// TIA Portal project "Box Sorting" (V18)

(* hardware
DEVICE "S7-1200 station_1"  S7-1200 Station
   slot 0: "Rack_0"  S7-1200 Rack  Rack  V1.0
   slot 1: "PLC_1"  CPU 1212C AC/DC/Rly  6ES7 212-1BE40-0XB0  V4.6
*)

// ===== PLC "PLC_1"  CPU 1212C AC/DC/Rly =====

VAR_GLOBAL   // PLC tag table "Default tag table"
   "Start" AT %I0.0 : Bool;
   "Auto Mode" AT %M0.0 : Bool;
   "Stop" AT %I0.1 : Bool;
   "PE_Low" AT %I0.2 : Bool;
   "PE_High" AT %I0.3 : Bool;
   "#Large Box" AT %M0.1 : Bool;
   "Motor1" AT %Q0.0 : Bool;
   "Solenoid_valve" AT %Q0.1 : Bool;
   "Motor2" AT %Q0.2 : Bool;
   "num_L" AT %MW2 : Int;
   "num_S" AT %MW4 : Int;
   "total_box" AT %MW6 : Int;
   "num_L_real" AT %MD8 : Real;
   "num_S_real" AT %MD12 : Real;
   "total_box_real" AT %MD16 : Real;
   "percent_large" AT %MD20 : Real;
   "percent_small" AT %MD24 : Real;
   "Emergency Stop" AT %I0.4 : Bool;
END_VAR

// folder: System blocks/Program resources

DATA_BLOCK "timerA_DB"   // DB1
{ S7_Optimized_Access := 'TRUE' }
AUTHOR : Simatic
FAMILY : IEC
NAME : IEC_TMR
VERSION : 1.0
// stored: InstanceOfName IEC_TIMER
"IEC_TIMER"
BEGIN
END_DATA_BLOCK

DATA_BLOCK "timerB_DB"   // DB2
{ S7_Optimized_Access := 'TRUE' }
AUTHOR : Simatic
FAMILY : IEC
NAME : IEC_TMR
VERSION : 1.0
// stored: InstanceOfName IEC_TIMER
"IEC_TIMER"
BEGIN
END_DATA_BLOCK

DATA_BLOCK "timerC_DB"   // DB3
{ S7_Optimized_Access := 'TRUE' }
AUTHOR : Simatic
FAMILY : IEC
NAME : IEC_TMR
VERSION : 1.0
// stored: InstanceOfName IEC_TIMER
"IEC_TIMER"
BEGIN
END_DATA_BLOCK

DATA_BLOCK "timerD_DB"   // DB4
{ S7_Optimized_Access := 'TRUE' }
AUTHOR : Simatic
FAMILY : IEC
NAME : IEC_TMR
VERSION : 1.0
// stored: InstanceOfName IEC_TIMER
"IEC_TIMER"
BEGIN
END_DATA_BLOCK

DATA_BLOCK "CounterL_DB"   // DB5
{ S7_Optimized_Access := 'TRUE' }
AUTHOR : Simatic
FAMILY : IEC
NAME : CNTR
VERSION : 1.0
// stored: InstanceOfName IEC_COUNTER
"IEC_COUNTER"
BEGIN
END_DATA_BLOCK

DATA_BLOCK "CounterS_DB"   // DB6
{ S7_Optimized_Access := 'TRUE' }
AUTHOR : Simatic
FAMILY : IEC
NAME : CNTR
VERSION : 1.0
// stored: InstanceOfName IEC_COUNTER
"IEC_COUNTER"
BEGIN
END_DATA_BLOCK

// folder: (top level)

ORGANIZATION_BLOCK "Main"   // OB1, LAD, ProgramCycle
TITLE = "Main Program Sweep (Cycle)"
{ S7_Optimized_Access := 'TRUE' }
VERSION : 0.1
   VAR_INPUT
      Initial_Call : Bool;   // Initial call of this OB
      Remanence : Bool;   // =True, if remanent data are available
   END_VAR
   VAR_TEMP
      "Large Box" : Bool;
      "Large Box_1" : Bool;
      "#Large Box" : Bool;
      "#Large Box_1" : Bool;
      Small_box : Bool;
      "#Large_box" : Bool;
      Large_box : Bool;
      division : Real;
   END_VAR
   VAR_TEMP   // added for the SCL form of the ladder/FBD networks
      _w1 : Bool;
      _w2 : Bool;
   END_VAR
BEGIN

REGION Network 1
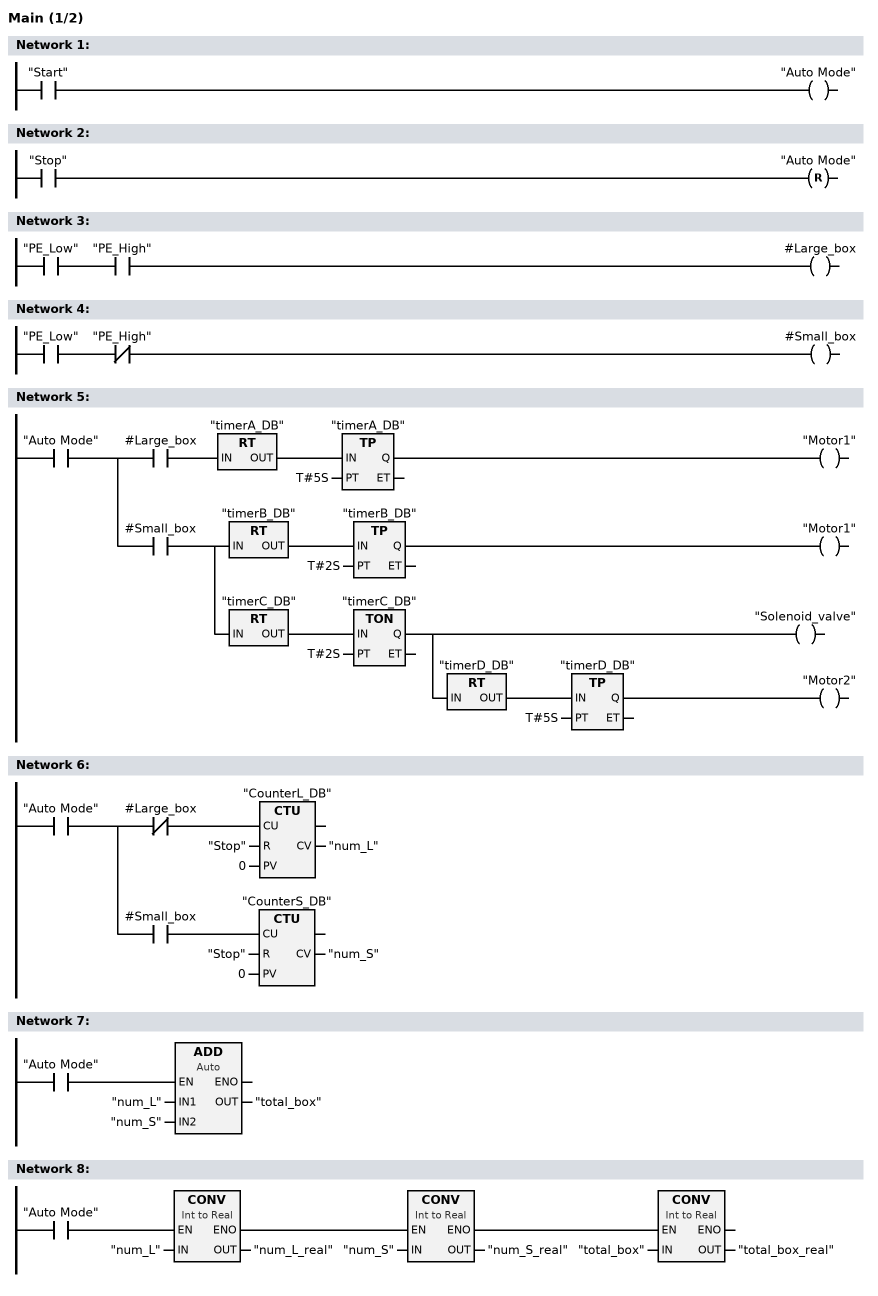
   RUNG wire#powerrail
      Contact( "Start" )
      Coil( "Auto Mode" )
   END_RUNG
   // the same network as SCL:
   "Auto Mode" := "Start";
END_REGION

REGION Network 2
   RUNG wire#powerrail
      Contact( "Stop" )
      R_Coil( "Auto Mode" )
   END_RUNG
   // the same network as SCL:
   IF "Stop" THEN "Auto Mode" := FALSE; END_IF;
END_REGION

REGION Network 3
   RUNG wire#powerrail
      Contact( "PE_Low" )
      Contact( "PE_High" )
      Coil( #Large_box )
   END_RUNG
   // the same network as SCL:
   #Large_box := "PE_Low" AND "PE_High";
END_REGION

REGION Network 4
   RUNG wire#powerrail
      Contact( "PE_Low" )
      I_Contact( "PE_High" )
      Coil( #Small_box )
   END_RUNG
   // the same network as SCL:
   #Small_box := "PE_Low" AND NOT "PE_High";
END_REGION

REGION Network 5
   #_w1 := "Auto Mode" AND #Large_box;
   IF #_w1 THEN RESET_TIMER("timerA_DB"); END_IF;
   "timerA_DB".TP(IN := #_w1, PT := T#5S);
   "Motor1" := "timerA_DB".Q;
   #_w2 := "Auto Mode" AND #Small_box;
   IF #_w2 THEN RESET_TIMER("timerB_DB"); END_IF;
   "timerB_DB".TP(IN := #_w2, PT := T#2S);
   "Motor1" := "timerB_DB".Q;
   IF #_w2 THEN RESET_TIMER("timerC_DB"); END_IF;
   "timerC_DB".TON(IN := #_w2, PT := T#2S);
   "Solenoid_valve" := "timerC_DB".Q;
   IF "timerC_DB".Q THEN RESET_TIMER("timerD_DB"); END_IF;
   "timerD_DB".TP(IN := "timerC_DB".Q, PT := T#5S);
   "Motor2" := "timerD_DB".Q;
END_REGION

REGION Network 6
   "CounterL_DB".CTU(CU := "Auto Mode" AND NOT #Large_box, R := "Stop", PV := 0, CV => "num_L");
   "CounterS_DB".CTU(CU := "Auto Mode" AND #Small_box, R := "Stop", PV := 0, CV => "num_S");
END_REGION

REGION Network 7
   RUNG wire#powerrail
      Contact( "Auto Mode" )
      Add(in1 := "num_L", in2 := "num_S", out => "total_box")
   END_RUNG
   // the same network as SCL:
   IF "Auto Mode" THEN "total_box" := "num_L" + "num_S"; END_IF;
END_REGION

REGION Network 8
   RUNG wire#powerrail
      Contact( "Auto Mode" )
      { S7_Templates := "[SrcType := Int, DestType := Real]" } Convert(in := "num_L", out => "num_L_real")
      { S7_Templates := "[SrcType := Int, DestType := Real]" } Convert(in := "num_S", out => "num_S_real")
      { S7_Templates := "[SrcType := Int, DestType := Real]" } Convert(in := "total_box", out => "total_box_real")
   END_RUNG
   // the same network as SCL:
   IF "Auto Mode" THEN
       "num_L_real" := INT_TO_REAL("num_L");
       "num_S_real" := INT_TO_REAL("num_S");
       "total_box_real" := INT_TO_REAL("total_box");
   END_IF;
END_REGION

REGION Network 9
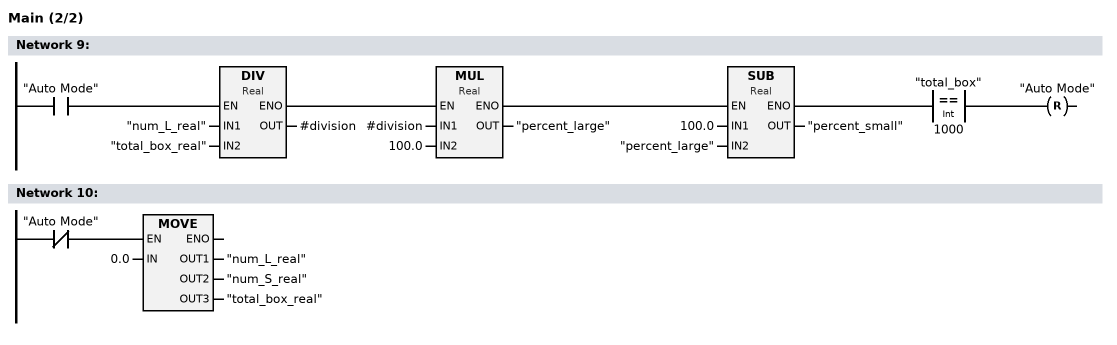
   RUNG wire#powerrail
      Contact( "Auto Mode" )
      { S7_Templates := "SrcType := Real" } Div(in1 := "num_L_real", in2 := "total_box_real", out => #division)
      { S7_Templates := "SrcType := Real" } Mul(in1 := #division, in2 := 100.0, out => "percent_large")
      { S7_Templates := "SrcType := Real" } Sub(in1 := 100.0, in2 := "percent_large", out => "percent_small")
      { S7_Templates := "SrcType := Int" } EQ_Contact(in1 := "total_box", in2 := 1000)
      R_Coil( "Auto Mode" )
   END_RUNG
   // the same network as SCL:
   IF "Auto Mode" THEN
       #division := "num_L_real" / "total_box_real";
       "percent_large" := #division * 100.0;
       "percent_small" := 100.0 - "percent_large";
   END_IF;
   IF "Auto Mode" AND ("total_box" = 1000) THEN "Auto Mode" := FALSE; END_IF;
END_REGION

REGION Network 10
   RUNG wire#powerrail
      I_Contact( "Auto Mode" )
      Move(in := 0.0, out1 => "num_L_real", out2 => "num_S_real", out3 => "total_box_real")
   END_RUNG
   // the same network as SCL:
   IF NOT "Auto Mode" THEN
       "num_L_real" := 0.0;
       "num_S_real" := 0.0;
       "total_box_real" := 0.0;
   END_IF;
END_REGION
END_ORGANIZATION_BLOCK